TYPE ST_Features :
STRUCT
	temp				: LREAL;
	cycle_time			: DINT;
	
	curr_mean			: LREAL;
	curr_peak			: LREAL;
	curr_range			: LREAL;
	curr_delta_max		: LREAL;
	curr_delta_idx		: LREAL;
	curr_std			: LREAL;
	                	
	vibe_mean			: LREAL;
	vibe_peak			: LREAL;
	vibe_range			: LREAL;
	vibe_delta_max		: LREAL;
	vibe_delta_idx		: LREAL;
	vibe_std			: LREAL;
END_STRUCT
END_TYPE

(* stored: Version 1.1.0.1, ProductVersion 3.1.4026.18
   DUT ST_Features: Id {4fb4ab5e-4e0f-4067-a6b0-e054b3a6ed07} *)
